FUNCTION TryConvert_UINT_TO_ULINT : BOOL
VAR_INPUT
	in : UINT;
	out : REFERENCE TO ULINT;
END_VAR

out := UINT_TO_ULINT(in);
TryConvert_UINT_TO_ULINT := TRUE;

END_FUNCTION

(* stored: Version 1.1.0.1, ProductVersion 3.1.4024.12
   POU TryConvert_UINT_TO_ULINT: Id {5ce88f7c-072e-4fce-a1f1-5e61020a0548}, SpecialFunc None *)
